// TIA Portal project "Project" (V16)

(* hardware
DEVICE "S7-1200 station_1"  S7-1200 Station
   slot 0: "Rack_0"  S7-1200 Rack  Rack  V1.0
   slot 1: "PLC_1"  CPU 1212C DC/DC/DC  6ES7 212-1AE40-0XB0  V4.4
DEVICE "PC-System_1"  SIMATIC PC station
   slot 0: "SIMATIC PC station"  Rail  SIMATIC PC-Station  V1.0
      slot 125: "Stationmanager"  Station_Manager  V6.0.4
   slot 1: "HMI_RT_1"  WinCC RT Advanced  6AV2 104-0xxxx-xxxx  16.0.0.0
      slot 33792: "Computer interface"  Host interface
   slot 2: "IE general_1"  IE General  IE_CP  V8.2.0
*)

// ===== PLC "PLC_1"  CPU 1212C DC/DC/DC =====

VAR_GLOBAL   // PLC tag table "Default tag table"
   "START" AT %I0.0 : Bool;
   "STOP" AT %I0.1 : Bool;
   "RUNNING" AT %M0.0 : Bool;
   "set home" AT %M0.1 : Bool;
   "Chai_Loi" AT %M0.2 : Bool;
   "enable" AT %Q0.4 : Bool;
   "ready" AT %I0.7 : Bool;
   "AxisOk" AT %Q0.5 : Bool;
   "Tag_1" AT %M6.0 : Bool;
   "Tag_2" AT %M30.0 : Bool;
   "m xilanh" AT %M30.1 : Bool;
   "swxilanh" AT %M30.2 : Bool;
   "Tag_3" AT %M30.3 : Bool;
   "Tag_4" AT %Q0.3 : Bool;
   "Tag_5" AT %M50.0 : Bool;
   "Tag_6" AT %M50.1 : Bool;
   "Tag_7" AT %M50.2 : Bool;
   "HOME" AT %MD8 : Real;
   "Tag_9" AT %M50.3 : Bool;
   "VITRI" AT %MD16 : Real;
   "TOCDO2" AT %MD4 : Real;
   "QUAYTHUAN" AT %M50.4 : Bool;
   "QUAYNGHICH" AT %M50.5 : Bool;
   "RESET" AT %I0.2 : Bool;
   "TIN_HIEU" AT %M50.6 : Bool;
   "Axis_1_Pulse" AT %Q0.0 : Bool;
   "Axis_1_Direction" AT %Q0.1 : Bool;
   "Xilanh" AT %Q0.2 : Bool;
END_VAR

DATA_BLOCK "Data_block_2"   // DB3
{ S7_Optimized_Access := 'FALSE' }
VERSION : 0.1
   VAR
      "SMU START" : Bool;
      "SMU STOP" : Bool;
      "SMU RESET" : Bool;
      "SMU SPEED" : Real := 2000.0;
      Static_2 : Int;
      Static_1 : Int;
      "TAY GAT" : Bool := false;
   END_VAR
BEGIN
END_DATA_BLOCK

DATA_BLOCK "Data_block_1"   // DB7
{ S7_Optimized_Access := 'FALSE' }
VERSION : 0.1
   VAR
      Enable : Bool;
      Reset : Bool;
      Halt : Bool;
      Home : Bool;
      MoveAbsolute : Bool;
      MoveRelative : Bool;
      JogForward : Bool;
      JogBackward : Bool;
      MoveVelocity : Bool;
      Position : Real := 6.0;
      Distance : Real := 6.0;
      Velocity : Real := 2000.0;
      stopmt : Bool;
   END_VAR
BEGIN
END_DATA_BLOCK

// folder: System blocks/Program resources

DATA_BLOCK "IEC_Timer_0_DB_1"   // DB16
{ S7_Optimized_Access := 'TRUE' }
AUTHOR : Simatic
FAMILY : IEC
NAME : IEC_TMR
VERSION : 1.0
// stored: InstanceOfName IEC_TIMER
"IEC_TIMER"
BEGIN
END_DATA_BLOCK

DATA_BLOCK "IEC_Timer_0_DB_3"   // DB17
{ S7_Optimized_Access := 'TRUE' }
AUTHOR : Simatic
FAMILY : IEC
NAME : IEC_TMR
VERSION : 1.0
// stored: InstanceOfName IEC_TIMER
"IEC_TIMER"
BEGIN
END_DATA_BLOCK

// folder: (top level)

DATA_BLOCK "Axis_1"   // DB1, Motion_DB
{ S7_Optimized_Access := 'TRUE' }
AUTHOR : SIMATIC
FAMILY : BasicMC
NAME : TO_PosAx
VERSION : 7.0
// stored: InstanceOfName TO_PositioningAxis
"TO_PositioningAxis"
BEGIN
   // Axis.EnableOutput_AddressCU = %Q0.0
   // Axis.DirectionOutputEnabledCU = TRUE
   // Axis.OnlinePtoModeCU = 16#0000_0002
   // Axis.SelectedChannel2EnumCU = %Q0.1
   // Axis.SelectedChannel1EnumCU = %Q0.0
   // Pulse.MinDeltaDeltaFrequencyCU = 0.004
   // Pulse.MaxDeltaDeltaFrequencyCU = 1.0E+10
   // Pulse.MinDeltaFrequencyCU = 0.005
   // Pulse.MaxDeltaFrequencyCU = 9.5E+9
   // Pulse.MinFrequencyCU = 1.0
   // Pulse.MaxFrequencyCU = 100000.0
   // Pulse.OutputSourceCU = 16#0000_0000
   // Axis.SelectPTO = 0
   // Axis.LengthUnit.LastDistance = -1
END_DATA_BLOCK

DATA_BLOCK "Axis_2"   // DB5, Motion_DB
{ S7_Optimized_Access := 'TRUE' }
AUTHOR : SIMATIC
FAMILY : BasicMC
NAME : TO_PosAx
VERSION : 7.0
// stored: InstanceOfName TO_PositioningAxis
"TO_PositioningAxis"
BEGIN
   // Axis.DirectionOutputEnabledCU = TRUE
   // Axis.OnlinePtoModeCU = 16#0000_0002
   // Axis.SelectedChannel2EnumCU = %Q0.3
   // Axis.SelectedChannel1EnumCU = %Q0.2
   // Pulse.MinDeltaDeltaFrequencyCU = 0.004
   // Pulse.MaxDeltaDeltaFrequencyCU = 1.0E+10
   // Pulse.MinDeltaFrequencyCU = 0.005
   // Pulse.MaxDeltaFrequencyCU = 9.5E+9
   // Pulse.MinFrequencyCU = 1.0
   // Pulse.MaxFrequencyCU = 100000.0
   // Pulse.OutputSourceCU = 16#0000_0000
   // Axis.SelectPTO = 1
   // Axis.OnlinePtoIndexCU = 1
   // Axis.LengthUnit.LastDistance = -1
END_DATA_BLOCK

ORGANIZATION_BLOCK "Main"   // OB1, LAD, ProgramCycle
TITLE = "Main Program Sweep (Cycle)"
{ S7_Optimized_Access := 'TRUE' }
VERSION : 0.1
   VAR_INPUT
      Initial_Call : Bool;   // Initial call of this OB
      Remanence : Bool;   // =True, if remanent data are available
   END_VAR
BEGIN

REGION Network 1
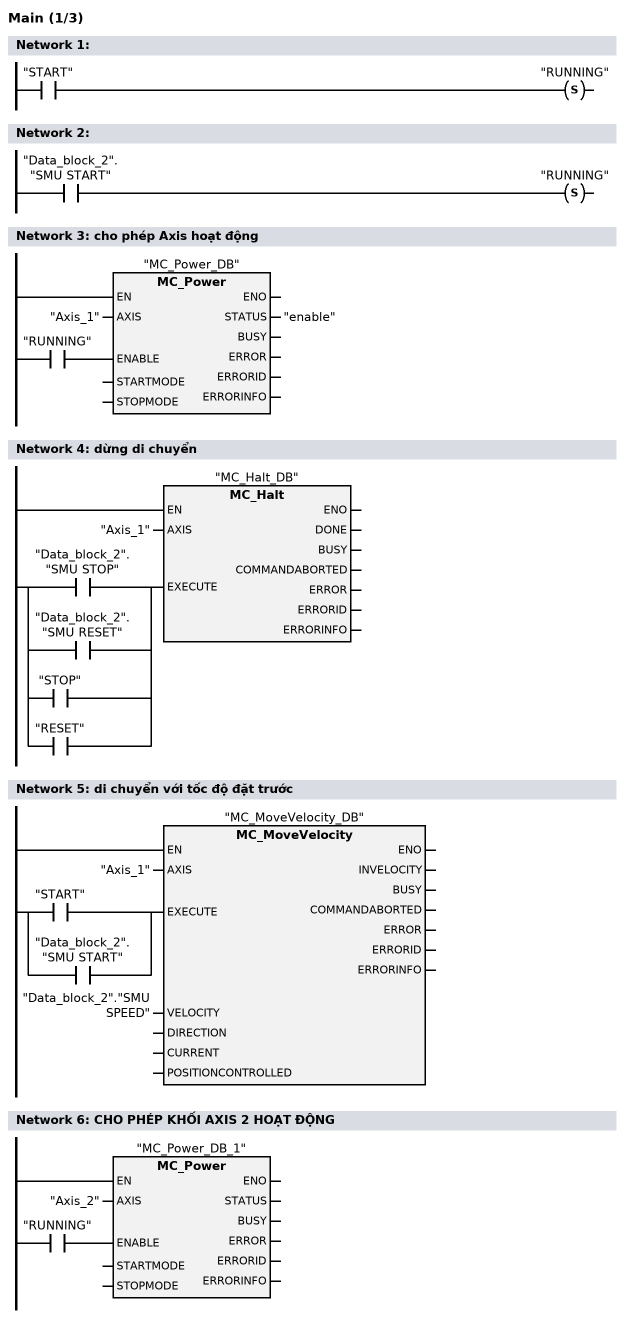
   RUNG wire#powerrail
      Contact( "START" )
      S_Coil( "RUNNING" )
   END_RUNG
   // the same network as SCL:
   IF "START" THEN "RUNNING" := TRUE; END_IF;
END_REGION

REGION Network 2
   RUNG wire#powerrail
      Contact( "Data_block_2"."SMU START" )
      S_Coil( "RUNNING" )
   END_RUNG
   // the same network as SCL:
   IF "Data_block_2"."SMU START" THEN "RUNNING" := TRUE; END_IF;
END_REGION

REGION Network 3: cho phép Axis hoạt động
   "MC_Power_DB"(Axis := "Axis_1", Enable := "RUNNING", Status => "enable");   // MC_Power
END_REGION

REGION Network 4: dừng di chuyển
   "MC_Halt_DB"(Axis := "Axis_1",   // MC_Halt
                Execute := "Data_block_2"."SMU STOP" OR "Data_block_2"."SMU RESET" OR "STOP" OR "RESET");
END_REGION

REGION Network 5: di chuyển với tốc độ đặt trước
   "MC_MoveVelocity_DB"(Axis := "Axis_1",   // MC_MoveVelocity
                        Execute := "START" OR "Data_block_2"."SMU START",
                        Velocity := "Data_block_2"."SMU SPEED");
END_REGION

REGION Network 6: CHO PHÉP KHỐI AXIS 2 HOẠT ĐỘNG
   "MC_Power_DB_1"(Axis := "Axis_2", Enable := "RUNNING");   // MC_Power
END_REGION

REGION Network 7: ĐẶT VỊ TRÍ HOME CHO TAY GẠT
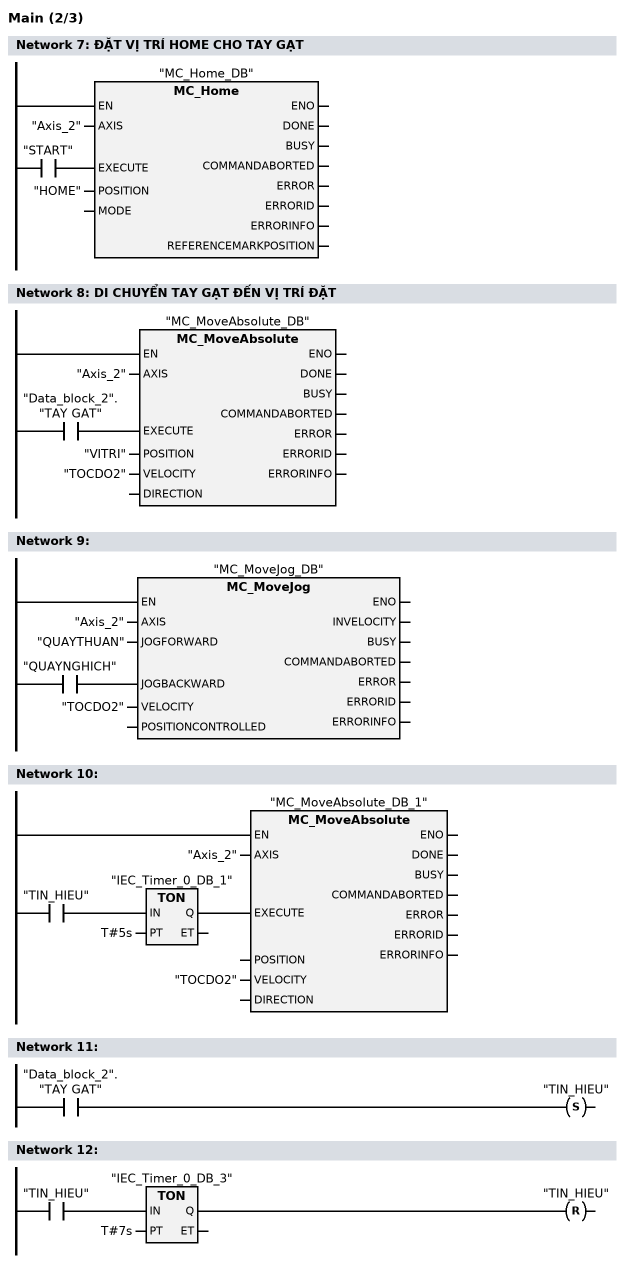
   "MC_Home_DB"(Axis := "Axis_2", Execute := "START", Position := "HOME");   // MC_Home
END_REGION

REGION Network 8: DI CHUYỂN TAY GẠT ĐẾN VỊ TRÍ ĐẶT
   "MC_MoveAbsolute_DB"(Axis := "Axis_2",   // MC_MoveAbsolute
                        Execute := "Data_block_2"."TAY GAT",
                        Position := "VITRI",
                        Velocity := "TOCDO2");
END_REGION

REGION Network 9
   "MC_MoveJog_DB"(Axis := "Axis_2",   // MC_MoveJog
                   JogForward := "QUAYTHUAN",
                   JogBackward := "QUAYNGHICH",
                   Velocity := "TOCDO2");
END_REGION

REGION Network 10
   "IEC_Timer_0_DB_1".TON(IN := "TIN_HIEU", PT := T#5s);
   "MC_MoveAbsolute_DB_1"(Axis := "Axis_2", Execute := "IEC_Timer_0_DB_1".Q, Velocity := "TOCDO2");   // MC_MoveAbsolute
END_REGION

REGION Network 11
   RUNG wire#powerrail
      Contact( "Data_block_2"."TAY GAT" )
      S_Coil( "TIN_HIEU" )
   END_RUNG
   // the same network as SCL:
   IF "Data_block_2"."TAY GAT" THEN "TIN_HIEU" := TRUE; END_IF;
END_REGION

REGION Network 12
   "IEC_Timer_0_DB_3".TON(IN := "TIN_HIEU", PT := T#7s);
   IF "IEC_Timer_0_DB_3".Q THEN "TIN_HIEU" := FALSE; END_IF;
END_REGION

REGION Network 13
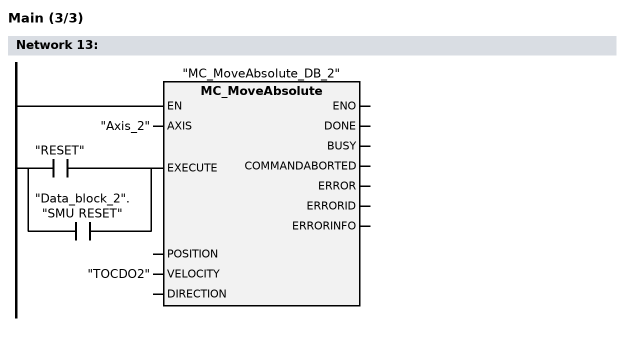
   "MC_MoveAbsolute_DB_2"(Axis := "Axis_2",   // MC_MoveAbsolute
                          Execute := "RESET" OR "Data_block_2"."SMU RESET",
                          Velocity := "TOCDO2");
END_REGION
END_ORGANIZATION_BLOCK

(* ===== HMI "HMI_RT_1" =====
system functions are stored by id; their names below are inferred from use
connection "HMI_Connection_1": ETHERNET, S7_1200_OMS

HMI tags "Default tag table"
   "M-START" : Bool = PLC "M-START" AT %M0.3, 1 s
   "M-STOP" : Bool = PLC "M-STOP" AT %M0.4, 1 s
   "RUNNING" : Bool = PLC RUNNING AT %M0.0, 1 s
   "Xilanh" : Bool = PLC Xilanh AT %Q0.2, 1 s
   "sensor" : Bool = PLC sensor AT %I0.3, 1 s
   "count" : Int = PLC count AT %MW204, 1 s
   "count-loi" : Int = PLC "count-loi" AT %MW205, 1 s
   "reset" : Bool = PLC Mreset AT %M0.5, 1 s
   "denxanh" : Bool = PLC denxanh AT %M1.0, 1 s
   "denvang" : Bool = PLC denvang AT %M1.3, 1 s
   "dendo" : Bool = PLC dendo AT %M1.1, 1 s
   "simuVTSP" : Int = PLC simuVTSP AT %MW214, 1 s
   "M-sensor" : Bool = PLC "M-sensor" AT %M10.1, 1 s
   "swxilanh" : Bool = PLC swxilanh AT %M30.2, 1 s
   "m xilanh" : Bool = PLC "m xilanh" AT %M30.1, 1 s

screen "Screen_1" 1024x1280
   TextField "Text field_1" at 102,19 size 632x22; Text 'ĐIỀU KHIỂN PHÂN LOẠI CHAI NƯỚC BỊ LỖI TRÊN S7-1200 VÀ WINCC TIA PORTAL'
   SymbolLibrary "Symbol library_1" at 191,199 size 574x73
      Appearance <- "RUNNING"
   SymbolLibrary "Symbol library_2" at 265,157 size 28x67
      HorizontalMovement <- "simuVTSP"
   Button "Button_1" at 23,61 size 79x38; TextOff 'START'
      on Press: SetBit("M-START")
      on Release: ResetBit("M-START")
   Button "Button_2" at 114,61 size 77x39; TextOff 'STOP'
      on Press: SetBit("M-STOP")
      on Release: ResetBit("M-STOP")
   Group "Group" at 504,70 size 123x91
   Group "Group_2" at 371,272 size 126x88
   SymbolLibrary "Symbol library_3" at 323,374 size 114x65
   TextField "Text field_2" at 333,441 size 101x22; Text 'Chai nước lỗi'
   SymbolLibrary "Symbol library_4" at 690,111 size 37x61
      Appearance <- "M-sensor"
   SymbolLibrary "Symbol library_5" at 694,271 size 118x68
   TextField "Text field_3" at 690,340 size 106x22; Text 'Chai nước đạt'
   IOField "I/O field_1" at 677,376 size 87x25; FormatPattern s99
      ProcessValue <- "count"
   TextField "Text field_4" at 762,378 size 50x22; Text '[chai]'
   IOField "I/O field_2" at 352,465 size 47x25; FormatPattern s99
      ProcessValue <- "count-loi"
   TextField "Text field_5" at 402,468 size 50x22; Text '[chai]'
   Button "Button_3" at 56,112 size 96x32; TextOff 'RESET'
      on Release: ResetBit("reset")
      on Press: SetBit("reset")
   Circle "Circle_1" at 28,155 size 42x42
      Appearance <- "denxanh"
   Circle "Circle_2" at 88,155 size 42x42
      Appearance <- "dendo"
   Circle "Circle_3" at 152,155 size 42x42
      Appearance <- "denvang"
   Switch "Switch_1" at 460,41 size 90x55; CaptionText 'Switch'; TextOff 'OFF'; TextOn 'ON'
      on SwitchOn: SetBit("swxilanh")
      on SwitchOff: ResetBit("swxilanh")
      ProcessValue <- "swxilanh"
   Group "Group_1" at 429,144 size 93x67
   Polyline "Polyline_2" at 441,144 size 81x59
      Visibility <- "m xilanh"

screen "Screen_2" 1024x1280
   TextField "Text field_1" at 362,29 size 15x22; Text 'Text'
   TextField "Text field_2" at 46,10 size 532x22; Text 'PHÂN LOẠI CHAI NƯỚC BỊ LỖI TRÊN S7-1200 VÀ WINCC TIA PORTAL'
   Button "Button_1" at 122,63 size 96x54; TextOff 'START'
      on Release: ResetBit("M-START")
      on Press: SetBit("M-START")
   Button "Button_2" at 262,62 size 98x54; TextOff 'STOP'
      on Release: ResetBit("M-STOP")
      on Press: SetBit("M-STOP")
   Button "Button_3" at 399,63 size 95x53; TextOff 'RESET'
      on Release: ResetBit("reset")
      on Press: SetBit("reset")
   Circle "Circle_1" at 150,148 size 56x56
      Appearance <- "denxanh"
   Circle "Circle_2" at 288,148 size 57x57
      Appearance <- "dendo"
   Circle "Circle_3" at 423,148 size 55x55
      Appearance <- "denvang"
   IOField "I/O field_2" at 149,287 size 47x25; FormatPattern s99
      ProcessValue <- "count-loi"
   TextField "Text field_5" at 204,289 size 50x22; Text '[chai]'
   TextField "Text field_3" at 126,256 size 152x22; Text 'SỐ CHAI NƯỚC LỖI'
   TextField "Text field_4" at 339,258 size 155x22; Text 'SỐ CHAI NƯỚC ĐẠT'
   IOField "I/O field_1" at 359,287 size 57x25; FormatPattern s99
      ProcessValue <- "count"
   TextField "Text field_6" at 431,289 size 50x22; Text '[chai]'
*)